{attribute 'GeneratedUsingTerminal: EK1100-0000-0018'}
{attribute addProperty BoxType "EK1100-0000-0018"}
{attribute addProperty Id "Beckhoff_EJ2xxxEK1122Beckhoff_EJ2xxxEK1122_536A68292A_0001_EJ2008_0000_0017EJ2008_E2806B9511A_0002_EJ2008_0000_0018EJ2008_E2806B9511A_0003_EJ2128_0000_0016EJ2128_E2806B9511A_0004_EJ2502_0000_0023EJ2502_8962CF717A_0005_EJ2502_0000_0024EJ2502_8962CF717A_0006_EJ2521_0224_0016EJ2521_E2FDA3CB52A_0007_EJ2522_0000_0022EJ2522_CC50E1AE64A_0008_EJ2809_0000_0017EJ2809_2B6483BD19A_0009_EJ2889_0000_0016EJ2889_2B6483BD19A_0010_EJ2889_0000_0017EJ2889_2B6483BD19"}
{attribute addProperty CRC "2660603287"}
{attribute addProperty Size "222"}
TYPE Beckhoff_EJ2xxx_9E959597 EXTENDS EK1100_1FC0878B :
STRUCT
	{attribute addProperty Name "Beckhoff_EJ2xxxEK1122"}
	{attribute addProperty PreviousPort "Beckhoff EJ2xxx : B"}
	Beckhoff_EJ2xxxEK1122 : Beckhoff_EJ2xxxEK1122_536A6829;
	{attribute addProperty Name "A_0001_EJ2008_0000_0017"}
	{attribute addProperty PreviousPort "Beckhoff EJ2xxxEK1122 : C"}
	A_0001_EJ2008_0000_0017 : EJ2008_E2806B95;
	{attribute addProperty Name "A_0002_EJ2008_0000_0018"}
	{attribute addProperty PreviousPort "A_0001(EJ2008-0000-0017) : B"}
	A_0002_EJ2008_0000_0018 : EJ2008_E2806B95;
	{attribute addProperty Name "A_0003_EJ2128_0000_0016"}
	{attribute addProperty PreviousPort "A_0002(EJ2008-0000-0018) : B"}
	A_0003_EJ2128_0000_0016 : EJ2128_E2806B95;
	{attribute addProperty Name "A_0004_EJ2502_0000_0023"}
	{attribute addProperty PreviousPort "A_0003(EJ2128-0000-0016) : B"}
	A_0004_EJ2502_0000_0023 : EJ2502_8962CF71;
	{attribute addProperty Name "A_0005_EJ2502_0000_0024"}
	{attribute addProperty PreviousPort "A_0004(EJ2502-0000-0023) : B"}
	A_0005_EJ2502_0000_0024 : EJ2502_8962CF71;
	{attribute addProperty Name "A_0006_EJ2521_0224_0016"}
	{attribute addProperty PreviousPort "A_0005(EJ2502-0000-0024) : B"}
	A_0006_EJ2521_0224_0016 : EJ2521_E2FDA3CB;
	{attribute addProperty Name "A_0007_EJ2522_0000_0022"}
	{attribute addProperty PreviousPort "A_0006(EJ2521-0224-0016) : B"}
	A_0007_EJ2522_0000_0022 : EJ2522_CC50E1AE;
	{attribute addProperty Name "A_0008_EJ2809_0000_0017"}
	{attribute addProperty PreviousPort "A_0007(EJ2522-0000-0022) : B"}
	A_0008_EJ2809_0000_0017 : EJ2809_2B6483BD;
	{attribute addProperty Name "A_0009_EJ2889_0000_0016"}
	{attribute addProperty PreviousPort "A_0008(EJ2809-0000-0017) : B"}
	A_0009_EJ2889_0000_0016 : EJ2889_2B6483BD;
	{attribute addProperty Name "A_0010_EJ2889_0000_0017"}
	{attribute addProperty PreviousPort "A_0009(EJ2889-0000-0016) : B"}
	A_0010_EJ2889_0000_0017 : EJ2889_2B6483BD;
END_STRUCT
END_TYPE

(* stored: Version 1.2.0.0, ProductVersion 3.1.4024.9
   DUT Beckhoff_EJ2xxx_9E959597: Id {a48637e9-1890-43ea-9041-34ab7de6f4c2} *)
